FUNCTION_BLOCK LTimeComparer EXTENDS Object IMPLEMENTS IComparer
VAR
	_ClassName : STRING := __POUNAME();
END_VAR

{attribute 'monitoring' := 'call'}
PROPERTY ClassName : STRING
GET
ClassName := _ClassName;
END_GET
END_PROPERTY

{attribute "object_name" := "Compare"}
METHOD Compare : COMPARISION_RESULT
VAR_INPUT
	left : GENERIC_VALUE;
	right : GENERIC_VALUE;
END_VAR
VAR
	leftPointer : POINTER TO LTIME; 
	rightPointer : POINTER TO LTIME; 
END_VAR
IF left.Address = 0 AND right.Address = 0 THEN
	Compare := COMPARISION_RESULT.EQUALS;
	RETURN;
END_IF

IF left.Address = 0 THEN
	Compare := COMPARISION_RESULT.LEFT_LESS_RIGHT;
	RETURN;	
END_IF

IF right.Address = 0 THEN
	Compare := COMPARISION_RESULT.LEFT_GREATER_RIGHT;
	RETURN;	
END_IF

leftPointer := left.Address;
rightPointer := right.Address;

IF leftPointer^ < rightPointer^ THEN
	Compare := COMPARISION_RESULT.LEFT_LESS_RIGHT;
ELSIF leftPointer^ > rightPointer^ THEN
	Compare := COMPARISION_RESULT.LEFT_GREATER_RIGHT;
ELSE
	Compare := COMPARISION_RESULT.EQUALS;	
END_IF
END_METHOD

{attribute 'monitoring' := 'call'}
PROPERTY Size : ULINT
GET
Size := XSIZEOF(THIS^);
END_GET
END_PROPERTY

END_FUNCTION_BLOCK

(* stored: Version 1.1.0.1
   POU LTimeComparer: Id {ace72394-daf6-4b9d-a33d-9a436c0a305e}, SpecialFunc None
   Property ClassName: Id {85665c3e-8f5e-44c8-b281-b80838358c8a}
   Get Get: Id {efcaf5c8-16fb-4602-8bb0-efa67641ae20}
   Method Compare: Id {b669a8e2-61ab-4523-b98f-4dc19e868351}
   Property Size: Id {589d987c-a708-4ea5-8f21-736c80a729d0}
   Get Get: Id {02fdeab4-5b77-4079-8ffc-c9e19327056c} *)
